// TIA Portal V19 export
DATA_BLOCK "ItemTimerwork"   // DB13
{ S7_Optimized_Access := 'TRUE' }
AUTHOR : FLA
FAMILY : UHT
VERSION : 1.0
// stored: AutoNumber false, MemoryReserve 0
   VAR RETAIN
      Y0101 : "ItemTimer_UDT";
      Y0103 : "ItemTimer_UDT";
      Y0104 : "ItemTimer_UDT";
      Y0109 : "ItemTimer_UDT";
      Y0111 : "ItemTimer_UDT";
      Y0112 : "ItemTimer_UDT";
      Y0113 : "ItemTimer_UDT";
      Y0114 : "ItemTimer_UDT";
      Y0115 : "ItemTimer_UDT";
      M0139 : "ItemTimer_UDT";
      Y0116 : "ItemTimer_UDT";
      Y0108 : "ItemTimer_UDT";
      Y0117 : "ItemTimer_UDT";
      Y0118 : "ItemTimer_UDT";
      Y0237 : "ItemTimer_UDT";
      Y0238 : "ItemTimer_UDT";
      Y0119 : "ItemTimer_UDT";
      Y0124 : "ItemTimer_UDT";
      Y0135_NOT_USED : "ItemTimer_UDT";
      Y0136_NOT_USED : "ItemTimer_UDT";
      Y0137_NOT_USED : "ItemTimer_UDT";
      Y0143 : "ItemTimer_UDT";
      Y0144_NOT_USED : "ItemTimer_UDT";
      Y0147 : "ItemTimer_UDT";
      Y0148 : "ItemTimer_UDT";
      Y0158 : "ItemTimer_UDT";
      Y0545 : "ItemTimer_UDT";
      PACK1 : "ItemTimer_UDT";
      PACK2 : "ItemTimer_UDT";
      PACK3 : "ItemTimer_UDT";
      PACK4 : "ItemTimer_UDT";
      AlarmLamp : "ItemTimer_UDT";
      AHV_CLOSED : "ItemTimer_UDT";
      AHV_HIGH_LEVEL : "ItemTimer_UDT";
      AHV_READY : "ItemTimer_UDT";
      AHV_SHUT_DOWN : "ItemTimer_UDT";
      AHV_STERILE : "ItemTimer_UDT";
      PROD_AVAILABLE : "ItemTimer_UDT";
      RINSE_READY : "ItemTimer_UDT";
      CAUSTIC_READY : "ItemTimer_UDT";
      ACID_READY : "ItemTimer_UDT";
      CIP_FILLER_ENABLE : "ItemTimer_UDT";
      WATER_PUMP : "ItemTimer_UDT";
      Y0901 : "ItemTimer_UDT";
      Y0902 : "ItemTimer_UDT";
      Y0903 : "ItemTimer_UDT";
      TANK_READY : "ItemTimer_UDT";
      TANK_OPEN : "ItemTimer_UDT";
      Y0904 : "ItemTimer_UDT";
      Y0905 : "ItemTimer_UDT";
      Y0906 : "ItemTimer_UDT";
      Y0907 : "ItemTimer_UDT";
      Y0908 : "ItemTimer_UDT";
      Y0909 : "ItemTimer_UDT";
      Y0910 : "ItemTimer_UDT";
      Y0911 : "ItemTimer_UDT";
      Y0912 : "ItemTimer_UDT";
      Q41_1 : "ItemTimer_UDT";
      CIP_Route : "ItemTimer_UDT";
      SIP_Steam : "ItemTimer_UDT";
      Product_Available : "ItemTimer_UDT";
      Barrier_Sterile : "ItemTimer_UDT";
      Product_Route : "ItemTimer_UDT";
      X0913 : "ItemTimer_UDT";
      V0930 : "ItemTimer_UDT";
      V0931 : "ItemTimer_UDT";
      spare2 : "ItemTimer_UDT";
      V0552 : "ItemTimer_UDT";
      V0934 : "ItemTimer_UDT";
      V0935 : "ItemTimer_UDT";
      V0940 : "ItemTimer_UDT";
      V0941 : "ItemTimer_UDT";
      V0942 : "ItemTimer_UDT";
      V0943 : "ItemTimer_UDT";
      V0944 : "ItemTimer_UDT";
      V0945 : "ItemTimer_UDT";
      M0940 : "ItemTimer_UDT";
      V1021 : "ItemTimer_UDT";
      V1023 : "ItemTimer_UDT";
      V1024 : "ItemTimer_UDT";
      V1025 : "ItemTimer_UDT";
      V1027 : "ItemTimer_UDT";
      V1083 : "ItemTimer_UDT";
      M0941 : "ItemTimer_UDT";
      V0936 : "ItemTimer_UDT";
   END_VAR
BEGIN
END_DATA_BLOCK
